FUNCTION AMSNETID_TO_STRING : STRING
VAR_INPUT
	AoeNetId 	: AMSNETID;
END_VAR
VAR
	Index		: INT := 0;
END_VAR

AMSNETID_TO_STRING := TO_STRING(AoeNetId[Index]);
FOR Index := 1 TO 5 DO
	AMSNETID_TO_STRING := CONCAT(AMSNETID_TO_STRING, '.');
	AMSNETID_TO_STRING := CONCAT(AMSNETID_TO_STRING, TO_STRING(AoeNetId[Index]));
END_FOR

END_FUNCTION

(* stored: Version 1.1.0.1, ProductVersion 3.1.4024.3
   POU AMSNETID_TO_STRING: Id {6fd44617-37fe-46df-a191-d0e661a56201}, SpecialFunc None *)
